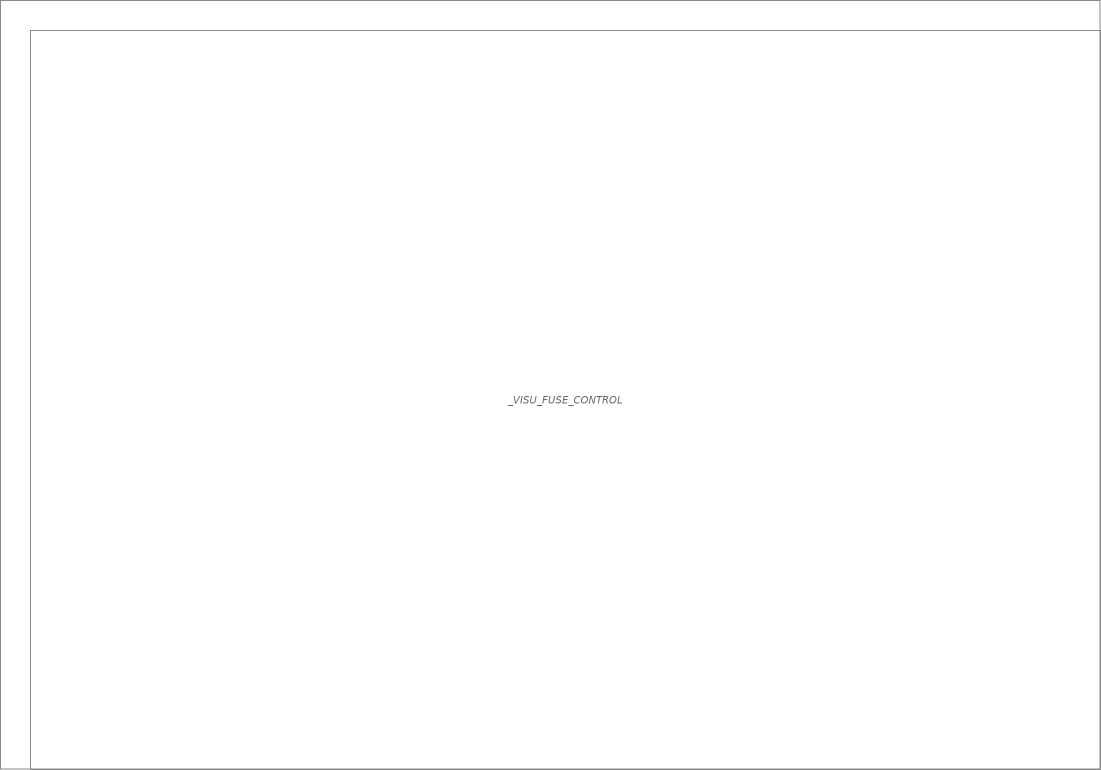
VISUALIZATION VISU_WeuControlStatus  // 1101x770
    Frame (30,30 1071x740)
        shows _VISU_FUSE_CONTROL(mInst := PRG_MACHINE.fbPowerControl)
END_VISUALIZATION

(* stored: Version 1.1.0.1, ProductVersion 3.1.4024.11
   Visu VISU_WeuControlStatus: Id {ad15781c-d5f4-43a1-a2aa-d1dabec89b9f} *)
